
FUNCTION CB_ge_time : BOOL


TITLE = ' Test Whether IN0 is greater than or equal to IN1 '
VERSION : '1.0'
AUTHOR  : CB
NAME    : ge_time
FAMILY  : TNI

VAR_INPUT
    IN0 : TIME;
    IN1 : TIME;
END_VAR

BEGIN

CB_ge_time := (IN0 >= IN1);

END_FUNCTION
